(* IEC 61131-3 sources: SJ_AGV/PLC/Standard_functions.4.4.0/Autoload, 3 files *)

(* ---- AutoLoadFailCodes.TYP ---- *)
[IEC_IEC_NORM]
TYPE
	AutoLoadFailCodes_T:
		STRUCT
			FailCode_OK						: word	:= 16#0000;
			FailCode_AGV_HalfLoad			: word	:= 16#0001;		(* Load is on the forks, but not fully. Manual handling and reset required! *)
			FailCode_OPNoSupport 			: word	:= 16#0002;
			FailCode_OpCancel 				: word	:= 16#0004;
			FailCode_InvalidOP 				: word	:= 16#0008;
			FailCode_AGVIsLoaded 			: word	:= 16#0010;
			FailCode_STNIsEmpty 			: word	:= 16#0020;
			FailCode_AGVIsNotLoaded			: word	:= 16#0040;
			FailCode_STNIsFull 				: word	:= 16#0080;
			FailCode_FirstPalletTooHigh		: word	:= 16#0100;
			FailCode_NoSecondPallet			: word	:= 16#0200;
			FailCode_SecondPalletTooLow		: word	:= 16#0400;
			FailCode_PalletOnInitialLift	: word	:= 16#0800;
			FailCode_NoPalletOnInitialLift	: word	:= 16#1000;
			FailCode_BatteryCharge			: word	:= 16#2000;
		END_STRUCT;
END_TYPE

(* ---- AUTOLOAD_FB.ST ---- *)
FUNCTION_BLOCK AUTOLOAD_FB
VAR_EXTERNAL
	(* IN *)
	NDC8: NDC8_T;
END_VAR

VAR_INPUT
	ForkMoving	: bool;
	ForkTarget	: bool;
END_VAR

VAR

	(* BCD Process *)
	BCDProcState : dint;
	BCDRetryTimes : int := 5;
	BCDReCompTimes : int := 5;
	BCDReadTimes : int;
	BCDCompTimes : int;

	TempBCD1_Int : Int;
	TempBCD1 : Word;

	(* Load/Unload Process *)
	LoadOpDone : LoadOpDone_FB;
	OperationFail : OperationFail_FB;

	AutoLoadFailCodes : AutoLoadFailCodes_T;
	OperationCode	: word;

	AutoLoadMainState : dint;

	BbxTrig_FT : F_trig;
	ExecDriveCommand_RT : R_Trig;
	FailTimerTON : TON;

	PreviousMainState,
	PreviousLoadState,
	PreviousUnLoadState,
	PreviousTravelDir,
	PreviousFailCode,
	PreviousForkHeight,
	FailCodeDint : dint;

	PreviousExecDriveCommand,
	PreviousCancelOperation,
	bbxtrigger			:bool;

	StepDelay : TON;
	BCDStepDelay : TON;

	TempErrorCode : DINT;

	BCD_ReadReq : BOOL;

	DebugBCD_1000_F : BOOL := FALSE;
	DebugBCD_1000_B : BOOL := FALSE;

	Debug_1000_F : BOOL := FALSE;
	Debug_1000_B : BOOL:= FALSE;
	Debug_2000_F : BOOL:= FALSE;
	Debug_2000_B : BOOL:= FALSE;

	LrErrCode : DINT;

	(*Wait Barcode Answer 2s*)

	WiatBardCodeAnser : TON;
END_VAR

VAR_OUTPUT
	StartLoad : bool;
	StartUnload : bool;
	StartCharge	: bool;
	Fail : bool;
END_VAR
(*
------------------------------------------------------------------------------------
 AUTOLOAD_SD
 -----------

 Description:
 Handles load operations. Output is 'Fork height'.
 If there is a cancel, LoadOpDone will be sent to the host with a failcode.

-------------------------------------------------------------------------------------*)

(* Set up variables to be used from NDC8 sources *)
OperationCode 		:= dint_to_word(NDC8.LoadOperation.OperationCode);				(* Value is decimal in vehicle, but hex in Layout designer! *)

if (NDC8.Automatic.CurrentOrderMode = 2 or NDC8.Automatic.CurrentOrderMode = 3) and AutoloadMainState <> 2000 then (*in Local mode Operation code need to calcuate for PLC*)
		IN_OPCD_Bit_LT_Ang0		:= word_to_bool(OperationCode and 1);
		IN_OPCD_Bit_LT_Ang90	:= word_to_bool(OperationCode and 2);
		IN_OPCD_Bit_LT_Ang180	:= word_to_bool(OperationCode and 8);
		IN_OPCD_Bit_LT_AngN90	:= word_to_bool(OperationCode and 4);

		IN_OPCD_Bit_LT_Right	:= word_to_bool(OperationCode and 16);
		IN_OPCD_Bit_LT_Left		:= word_to_bool(OperationCode and 32);

		IN_OPCD_Bit_LT_Load 	:= word_to_bool(OperationCode and 256);
		IN_OPCD_Bit_LT_Unload	:= word_to_bool(OperationCode and 512);

		IN_OPCD_Bit_LT_PowOff	:= word_to_bool(OperationCode and 1024);
		IN_OPCD_Bit_LT_Charge	:= word_to_bool(OperationCode and 4096);

elsif NDC8.Automatic.CurrentOrderMode = 1 and AutoloadMainState <> 2000 then (*in Host mode Operation code need to calcuate for PLC*)
		IN_OPCD_Bit_LT_Ang0		:= word_to_bool(OperationCode and 16);
		IN_OPCD_Bit_LT_Ang90	:= word_to_bool(OperationCode and 32);
		IN_OPCD_Bit_LT_Ang180	:= word_to_bool(OperationCode and 64);
		IN_OPCD_Bit_LT_AngN90	:= word_to_bool(OperationCode and 128);

		IN_OPCD_Bit_LT_Right	:= word_to_bool(OperationCode and 1);
		IN_OPCD_Bit_LT_Left		:= word_to_bool(OperationCode and 2);

		IN_OPCD_Bit_LT_Load 	:= word_to_bool(OperationCode and 4096);
		IN_OPCD_Bit_LT_Unload	:= word_to_bool(OperationCode and 8192);

		IN_OPCD_Bit_Cmd_EnaEmg	:= word_to_bool(OperationCode and 256);

		IN_OPCD_Bit_LT_PowOff	:= word_to_bool(OperationCode and 16384);

		IN_OPCD_Bit_LT_Charge	:= word_to_bool(OperationCode and 32768);

else
		OperationCode := 0;
		InProc_OperationCode := 0;
end_if;

(*Check Str_EnaPB *)
if NDC8.OMPLC.Phase - 4 >= 0 then
	PLC_TX01_Bit_STr_EnaPB := TRUE;
else
	PLC_TX01_Bit_STr_EnaPB := FALSE;
end_if;

(* BCD Process *)
if NDC8.Automatic.CurrentOrderMode = 1 and PLC_RX01_Bit_Load_i = TRUE then

	case BCDProcState of
	0: (* Check BCD Req *)
		OM_PLC_Word2 := INT_TO_WORD(NDC8.OMPLC.Stop_OM);

		BCDReadTimes := 0;
		BCDCompTimes := 0;

		if BCD_ReadReq = TRUE and OM_PLC_W2_Bit_BCD_NoRead = FALSE then
			BCDProcState := 1;
		elsif BCD_ReadReq = TRUE and OM_PLC_W2_Bit_BCD_NoRead = TRUE then
			BCD_ReadReq := FALSE;
		elsif OM_PLC_W2_Bit_BCD_NoRead = TRUE then
			BCDProcState := 0;
		elsif OM_PLC_W2_Bit_BCD_Init = TRUE and OM_PLC_W2_Bit_BCD_NoRead = FALSE then
			BCDProcState := 1;
		elsif OM_PLC_W2_Bit_BCD_setReq = TRUE and OM_PLC_W2_Bit_BCD_NoRead = FALSE then
			BCDProcState := 1;
		end_if;

		NDC8.OMPLC.Stop_OM := WORD_TO_INT(OM_PLC_Word2);
	1: (*Clear BCD Req*)
		StopByBCD := TRUE;
		PLC_TX04_Bit_BCD_Clr := true;
		PLC_TX04_Bit_BCD_Req := false;

		OM_PLC_Word2 := INT_TO_WORD(NDC8.OMPLC.Stop_OM);
			OM_PLC_W2_Bit_BCD_setOK := FALSE;
			OM_PLC_W2_Bit_Set_Result := FALSE;
			OM_PLC_W2_Bit_Err_Comp := FALSE;
			OM_PLC_W2_Bit_Err_BCR := FALSE;
		NDC8.OMPLC.Stop_OM := WORD_TO_INT(OM_PLC_Word2);

		if	not PLC_RX06_Bit_BCD_OK
			and not PLC_RX06_Bit_NoRead_NG
			and not PLC_RX06_Bit_BCRHard_NG
			and not PLC_RX06_Bit_BCRData_NG
			and not PLC_RX06_Bit_BCRInit_NG
			and not PLC_RX06_Bit_BCRComm_NG then

			BCDProcState := 2;
		end_if;

	2: (*Set BCD Req*)
		PLC_TX04_Bit_BCD_Clr := false;
		PLC_TX04_Bit_BCD_Req := true;
		WiatBardCodeAnser(IN := PLC_TX04_Bit_BCD_Req , PT:= t#2s);
		BCDReadTimes := BCDReadTimes + 1;
	IF WiatBardCodeAnser.Q = TRUE THEN
		if PLC_RX06_Bit_BCD_OK
			and not PLC_RX06_Bit_NoRead_NG
			and not PLC_RX06_Bit_BCRHard_NG
			and not PLC_RX06_Bit_BCRData_NG
			and not PLC_RX06_Bit_BCRInit_NG
			and not PLC_RX06_Bit_BCRComm_NG then
			BCDReadTimes := 0;

			BCDProcState := 3;

		elsif 	PLC_RX06_Bit_NoRead_NG
				or PLC_RX06_Bit_BCRHard_NG
				or PLC_RX06_Bit_BCRData_NG
				or PLC_RX06_Bit_BCRInit_NG
				or PLC_RX06_Bit_BCRComm_NG then

			if BCDReadTimes >= BCDRetryTimes then
				OM_PLC_Word2 := INT_TO_WORD(NDC8.OMPLC.Stop_OM);
					OM_PLC_W2_Bit_Err_BCR := TRUE;
					OM_PLC_W2_Bit_Set_Result := TRUE;
				NDC8.OMPLC.Stop_OM := WORD_TO_INT(OM_PLC_Word2);
				BCDProcState := 1000;
			else
				BCDProcState := 1;
			end_if;
		end_if;
	END_IF;
	3: (*BCD Compare*)
		WiatBardCodeAnser(IN := FALSE);
		TempBCD1_Int := WORD_TO_INT(PLC_RX_Word9_STw_BCD1);(* - 16#D00*);
		TempBCD1 := INT_TO_WORD(TempBCD1_Int);

		BCDCompTimes := BCDCompTimes + 1;

		if 	PLC_TX_Word14_STr_BCD3 = PLC_RX_Word7_STw_BCD3
			and PLC_TX_Word15_STr_BCD2 = PLC_RX_Word8_STw_BCD2
			and PLC_TX_Word16_STr_BCD1 = PLC_RX_Word9_STw_BCD1 then
			BCDProcState := 4; (* Compare Complete *)
			BCDCompTimes := 0;

		else

			if BCDCompTimes >= BCDReCompTimes then
				OM_PLC_Word2 := INT_TO_WORD(NDC8.OMPLC.Stop_OM);
					OM_PLC_W2_Bit_Err_Comp := TRUE;
					OM_PLC_W2_Bit_Set_Result := TRUE;
				NDC8.OMPLC.Stop_OM := WORD_TO_INT(OM_PLC_Word2);
				BCDProcState := 1000;
			else
				BCDProcState := 1;
			end_if;

		end_if;

	4:
		OM_PLC_Word2 := INT_TO_WORD(NDC8.OMPLC.Stop_OM);
			OM_PLC_W2_Bit_BCD_setOK := TRUE;
			OM_PLC_W2_Bit_Set_Result := TRUE;
		NDC8.OMPLC.Stop_OM := WORD_TO_INT(OM_PLC_Word2);
		BCDProcState := 1000;

	1000: (*Reset*)

		if DebugBCD_1000_F = FALSE then
			if DebugBCD_1000_B = FALSE then
				BCDProcState := 0;
			end_if;
			BCDReadTimes := 0;
			BCDCompTimes := 0;

			BCD_ReadReq := FALSE;
			StopByBCD := FALSE;
			BCDStepDelay(IN:= FALSE);

			OM_PLC_Word2 := INT_TO_WORD(NDC8.OMPLC.Stop_OM);
				OM_PLC_W2_Bit_BCD_setReq := FALSE;
				OM_PLC_W2_Bit_BCD_Init := FALSE;
			NDC8.OMPLC.Stop_OM := WORD_TO_INT(OM_PLC_Word2);
		end_if;

	end_case;
end_if;

Case AutoloadMainState of

(**** Wait for AutoLoad Start Flag - Operation Code > 0 ****)
	0:

		OM_PLC_Word2 := INT_TO_WORD(NDC8.OMPLC.Stop_OM);

		PLC_TX_Word2 := 0;

		PLC_TX02_Bit_STr_DepoST := FALSE;
		PLC_TX02_Bit_STr_ShutEQ := FALSE;
		PLC_TX04_Bit_Cancel_ST := FALSE;
		StepDelay(IN := FALSE);
		if g_ErrorCode = 0 and PLC_RX01_Bit_EnableLD_i = TRUE then
			if OperationCode > 0 then
				AutoloadMainState := 10;
			elsif NDC8.LocalOrder.OrderEN then
				AutoloadMainState := 10;
			end_if;
		end_if;

(**** Load operations ****)
	10:
		BCD_ReadReq := FALSE;
		INPUT.AutoLoadDone := FALSE;
		if 	IN_OPCD_Bit_LT_Load then	(* Load *)
			AutoloadMainState := 20;
		elsif 	IN_OPCD_Bit_LT_Unload then	(* Unload *)
			AutoloadMainState := 30;
		elsif 	IN_OPCD_Bit_LT_Charge then	(* Charge battery *)
			AutoloadMainState := 40;
		elsif	IN_OPCD_Bit_LT_PowOff then	(* Power off *)
			AutoloadMainState := 50;
		elsif NDC8.LocalOrder.OpCode = 0 then
			AutoloadMainState := 60;		(* Move no OP Code *)
		end_if;

(* Pick up load *)
	20:	(*Check Vehicle on Target Station*)

		OM_PLC_Word2 := INT_TO_WORD(NDC8.OMPLC.Stop_OM);

			OM_PLC_W2_Bit_SetT10Terr := FALSE;
			OM_PLC_W2_Bit_SetCondErr := FALSE;
			OM_PLC_W2_Bit_SetT30TErr := FALSE;
			OM_PLC_W2_Bit_SetHOErr := FALSE;

		NDC8.OMPLC.Stop_OM := WORD_TO_INT(OM_PLC_Word2);

		if g_ErrorCode <> 0 then
			AutoloadMainState := 999;
		else
			StartLoad := true;
			if NDC8.LoadDocking.OnTarget = TRUE and PLC_RX01_Bit_EnableLD_i = TRUE then
				AutoloadMainState := 21;
			elsif NDC8.LoadDocking.OnTarget = TRUE and PLC_RX01_Bit_EnableLD_i = FALSE then
				AutoloadMainState := 148;
			elsif InProc_OperationCode = 0 then
				AutoloadMainState := 145;
			end_if;
		end_if;

	21:(*Check Robot Load status*)
		StopLoadOP := TRUE;
		if g_ErrorCode <> 0 then
			AutoloadMainState := 999;
		else
			if PLC_RX01_Bit_Load_i = true then
				AutoloadMainState := 148;
			elsif NDC8.SDIO.DigitalInput12_EMO = FALSE then
				AutoloadMainState := 133;
			else
				AutoloadMainState := 22;
			end_if;
		end_if;

	22:(*Set OpCode to PLC*)

		if g_ErrorCode <> 0 then
			AutoloadMainState := 999;
		else
			PLC_TX02_Bit_STr_Ang0	:= IN_OPCD_Bit_LT_Ang0;
			PLC_TX02_Bit_STr_Ang90	:= IN_OPCD_Bit_LT_Ang90;
			PLC_TX02_Bit_STr_Ang180	:= IN_OPCD_Bit_LT_Ang180;
			PLC_TX02_Bit_STr_AngN90	:= IN_OPCD_Bit_LT_AngN90;

			PLC_TX02_Bit_STr_Right	:= IN_OPCD_Bit_LT_Right;
			PLC_TX02_Bit_STr_Left	:= IN_OPCD_Bit_LT_Left;

			PLC_TX02_Bit_STr_Load 	:= IN_OPCD_Bit_LT_Load;
			PLC_TX02_Bit_STr_Unload	:= IN_OPCD_Bit_LT_Unload;

			PLC_TX02_Bit_STr_DepoST := NDC8.PointTrigger.Bit0_DepoST_Att;
			PLC_TX02_Bit_STr_ShutEQ := NDC8.PointTrigger.Bit1_ShutEQ_Att;
			PLC_TX04_Bit_Cancel_ST := not IN_OPCD_Bit_Cmd_EnaEmg;

			if (PLC_TX02_Bit_STr_Ang0 = TRUE and PLC_TX02_Bit_STr_Ang90 = TRUE)
				or (PLC_TX02_Bit_STr_Ang0 = TRUE and PLC_TX02_Bit_STr_Ang180 = TRUE)
				or (PLC_TX02_Bit_STr_Ang0 = TRUE and PLC_TX02_Bit_STr_AngN90 = TRUE)
				or (PLC_TX02_Bit_STr_Ang90 = TRUE and PLC_TX02_Bit_STr_Ang180 = TRUE)
				or (PLC_TX02_Bit_STr_Ang90 = TRUE and PLC_TX02_Bit_STr_AngN90 = TRUE)
				or (PLC_TX02_Bit_STr_Ang180 = TRUE and PLC_TX02_Bit_STr_AngN90 = TRUE)
				or (PLC_TX02_Bit_STr_Right = TRUE and PLC_TX02_Bit_STr_Left = TRUE)
				or (PLC_TX02_Bit_STr_Load = TRUE and PLC_TX02_Bit_STr_Unload = TRUE) then

				if NDC8.Automatic.CurrentOrderMode = 1 then
					AutoloadMainState := 150;
				elsif NDC8.Automatic.CurrentOrderMode = 2 or NDC8.Automatic.CurrentOrderMode = 3 then
					AutoloadMainState := 152;
				end_if;

			elsif 	PLC_TX02_Bit_STr_Ang0 = FALSE
					and PLC_TX02_Bit_STr_Ang90 = FALSE
					and PLC_TX02_Bit_STr_Ang180 = FALSE
					and PLC_TX02_Bit_STr_AngN90 = FALSE then
					AutoloadMainState := 145;

			elsif	PLC_TX02_Bit_STr_Right = FALSE
					and PLC_TX02_Bit_STr_Left = FALSE then
					AutoloadMainState := 145;

			elsif	PLC_TX02_Bit_STr_Load = FALSE
					and PLC_TX02_Bit_STr_Unload = FALSE then
					AutoloadMainState := 145;

			else
				AutoloadMainState := 23;
			end_if;
		end_if;

	23:(*Wait PLC Processing*)
		if g_ErrorCode <> 0 then
			AutoloadMainState := 999;
		else
			if INPUT.Auto = FALSE then
				AutoloadMainState := 998;
			elsif NDC8.SDIO.DigitalInput12_EMO = FALSE then
				AutoloadMainState := 133;
			elsif PLC_RX01_Bit_LDErr_i then
				AutoloadMainState := 148;
			elsif PLC_RX_Word10_STw_ILEr <> 0 then (* Interlock (8I/8O) Proc *)

				OM_PLC_Word2 := INT_TO_WORD(NDC8.OMPLC.Stop_OM);

				case PLC_RX_Word10_STw_ILEr of
				1:
					OM_PLC_W2_Bit_SetT10Terr := TRUE;
					AutoloadMainState := 900;
				2:
					OM_PLC_W2_Bit_SetCondErr := TRUE;
					AutoloadMainState := 900;
				3:
					OM_PLC_W2_Bit_SetT30TErr := TRUE;
					AutoloadMainState := 900;
				4:
					OM_PLC_W2_Bit_SetHOErr := TRUE;
					AutoloadMainState := 900;
				5:
					OM_PLC_W2_Bit_SetHOErr := TRUE;
					AutoloadMainState := 900;

				end_case;

				NDC8.OMPLC.Stop_OM := WORD_TO_INT(OM_PLC_Word2);

			elsif PLC_RX01_Bit_LDDone_i then
				PLC_TX_Word2 := 0;
				PLC_TX02_Bit_STr_DepoST := FALSE;
				PLC_TX02_Bit_STr_ShutEQ := FALSE;
				PLC_TX04_Bit_Cancel_ST := FALSE;
			IF NDC8.Automatic.CurrentOrderMode = 1 THEN
				StopByBCD := TRUE;
			END_IF;
				BCD_ReadReq := TRUE;

				AutoloadMainState := 1000;
			end_if;
		end_if;

(* Drop off load *)
	30:	(*Check Vehicle on Target Station*)

		OM_PLC_Word2 := INT_TO_WORD(NDC8.OMPLC.Stop_OM);

			OM_PLC_W2_Bit_SetT10Terr := FALSE;
			OM_PLC_W2_Bit_SetCondErr := FALSE;
			OM_PLC_W2_Bit_SetT30TErr := FALSE;
			OM_PLC_W2_Bit_SetHOErr := FALSE;

		NDC8.OMPLC.Stop_OM := WORD_TO_INT(OM_PLC_Word2);

		if g_ErrorCode <> 0 then
			AutoloadMainState := 999;
		else
			StartUnload := true;

			if NDC8.LoadDocking.OnTarget = TRUE and PLC_RX01_Bit_EnableLD_i = TRUE then
				AutoloadMainState := 31;
			elsif NDC8.LoadDocking.OnTarget = TRUE and PLC_RX01_Bit_EnableLD_i = FALSE then
				AutoloadMainState := 149;
			end_if;
		end_if;

	31:(*Check Robot Load status*)
		StopLoadOP := TRUE;

		if g_ErrorCode <> 0 then
			AutoloadMainState := 999;
		else
			if PLC_RX01_Bit_Load_i = false then
				AutoloadMainState := 149;
			elsif NDC8.SDIO.DigitalInput12_EMO = FALSE then
				AutoloadMainState := 133;
			else
				AutoloadMainState := 32;
			end_if;
		end_if;

	32: (*Set OpCode to PLC*)

		if g_ErrorCode <> 0 then
			AutoloadMainState := 999;
		else
			PLC_TX02_Bit_STr_Ang0	:= IN_OPCD_Bit_LT_Ang0;
			PLC_TX02_Bit_STr_Ang90	:= IN_OPCD_Bit_LT_Ang90;
			PLC_TX02_Bit_STr_Ang180	:= IN_OPCD_Bit_LT_Ang180;
			PLC_TX02_Bit_STr_AngN90	:= IN_OPCD_Bit_LT_AngN90;

			PLC_TX02_Bit_STr_Right	:= IN_OPCD_Bit_LT_Right;
			PLC_TX02_Bit_STr_Left	:= IN_OPCD_Bit_LT_Left;

			PLC_TX02_Bit_STr_Load 	:= IN_OPCD_Bit_LT_Load;
			PLC_TX02_Bit_STr_Unload	:= IN_OPCD_Bit_LT_Unload;

			PLC_TX02_Bit_STr_DepoST := NDC8.PointTrigger.Bit0_DepoST_Att;
			PLC_TX02_Bit_STr_ShutEQ := NDC8.PointTrigger.Bit1_ShutEQ_Att;

			PLC_TX04_Bit_Cancel_ST := not IN_OPCD_Bit_Cmd_EnaEmg;

			if (PLC_TX02_Bit_STr_Ang0 = TRUE and PLC_TX02_Bit_STr_Ang90 = TRUE)
				or (PLC_TX02_Bit_STr_Ang0 = TRUE and PLC_TX02_Bit_STr_Ang180 = TRUE)
				or (PLC_TX02_Bit_STr_Ang0 = TRUE and PLC_TX02_Bit_STr_AngN90 = TRUE)
				or (PLC_TX02_Bit_STr_Ang90 = TRUE and PLC_TX02_Bit_STr_Ang180 = TRUE)
				or (PLC_TX02_Bit_STr_Ang90 = TRUE and PLC_TX02_Bit_STr_AngN90 = TRUE)
				or (PLC_TX02_Bit_STr_Ang180 = TRUE and PLC_TX02_Bit_STr_AngN90 = TRUE)
				or (PLC_TX02_Bit_STr_Right = TRUE and PLC_TX02_Bit_STr_Left = TRUE)
				or (PLC_TX02_Bit_STr_Load = TRUE and PLC_TX02_Bit_STr_Unload = TRUE) then

				if NDC8.Automatic.CurrentOrderMode = 1 then
					AutoloadMainState := 150;
				elsif NDC8.Automatic.CurrentOrderMode = 2 or NDC8.Automatic.CurrentOrderMode = 3 then
					AutoloadMainState := 152;
				end_if;

			elsif 	PLC_TX02_Bit_STr_Ang0 = FALSE
					and PLC_TX02_Bit_STr_Ang90 = FALSE
					and PLC_TX02_Bit_STr_Ang180 = FALSE
					and PLC_TX02_Bit_STr_AngN90 = FALSE then
					AutoloadMainState := 145;

			elsif	PLC_TX02_Bit_STr_Right = FALSE
					and PLC_TX02_Bit_STr_Left = FALSE then
					AutoloadMainState := 145;

			elsif	PLC_TX02_Bit_STr_Load = FALSE
					and PLC_TX02_Bit_STr_Unload = FALSE then
					AutoloadMainState := 145;

			else
				AutoloadMainState := 33;
			end_if;
		end_if;

	33: (*Wait PLC Processing*)
		if g_ErrorCode <> 0 then
				AutoloadMainState := 999;
		else
			if INPUT.Auto = FALSE then
				AutoloadMainState := 998;
			elsif NDC8.SDIO.DigitalInput12_EMO = FALSE then
				AutoloadMainState := 133;
			elsif PLC_RX01_Bit_LDErr_i then
				AutoloadMainState := 149;
			elsif PLC_RX_Word10_STw_ILEr <> 0 then (* Interlock (8I/8O) Proc *)

				OM_PLC_Word2 := INT_TO_WORD(NDC8.OMPLC.Stop_OM);

				case PLC_RX_Word10_STw_ILEr of
				1:
					OM_PLC_W2_Bit_SetT10Terr := TRUE;
					AutoloadMainState := 900;
				2:
					OM_PLC_W2_Bit_SetCondErr := TRUE;
					AutoloadMainState := 900;
				3:
					OM_PLC_W2_Bit_SetT30TErr := TRUE;
					AutoloadMainState := 900;
				4:
					OM_PLC_W2_Bit_SetHOErr := TRUE;
					AutoloadMainState := 900;
				5:
					OM_PLC_W2_Bit_SetHOErr := TRUE;
					AutoloadMainState := 900;

				end_case;

				NDC8.OMPLC.Stop_OM := WORD_TO_INT(OM_PLC_Word2);

			elsif PLC_RX01_Bit_LDDone_i then
				PLC_TX_Word2 := 0;
				PLC_TX02_Bit_STr_DepoST := FALSE;
				PLC_TX02_Bit_STr_ShutEQ := FALSE;
				PLC_TX04_Bit_Cancel_ST := FALSE;
				AutoloadMainState := 1000;
			end_if;
		end_if;

(* Charge the battery Local Order *)
	40:
		if g_ErrorCode <> 0 then
			AutoloadMainState := 999;
		else
			if NDC8.LoadDocking.OnTarget = TRUE then
				(* Wait Charger InPosition *)

				(* Check Charge Idle*)
				if PLC_RX01_Bit_ChrgIdle then
					AutoloadMainState := 41;
				end_if;

			end_if;
		end_if;

	41:(* Check OpCode and wait 10sec*)

		if g_ErrorCode <> 0 then
			AutoloadMainState := 49;
		else
			if INPUT.Auto = FALSE then
				AutoloadMainState := 49;
			end_if;

			if NDC8.PointTrigger.Bit9_Chrg_Right = TRUE or NDC8.PointTrigger.Bit10_Chrg_Left = TRUE  then
				StopCharge := TRUE;

				OM_PLC_Word2 := INT_TO_WORD(NDC8.OMPLC.Stop_OM);

				if (NDC8.Automatic.CurrentOrderMode = 1 and OM_PLC_W2_Bit_Set_LowTS) or NDC8.Automatic.CurrentOrderMode <> 1 then
					AutoloadMainState := 42;
				end_if;
			else
				;(*OP Error*)
			end_if;
		end_if;

	42:

		if g_ErrorCode <> 0 then
			AutoloadMainState := 49;
		else
			if INPUT.Auto = FALSE then
				AutoloadMainState := 49;
			end_if;
			IF NDC8.PointTrigger.Bit9_Chrg_Right = TRUE and NDC8.PointTrigger.Bit10_Chrg_Left = FALSE  then
				PLC_TX04_Bit_ChrgCmdR_A := TRUE;
				PLC_TX04_Bit_ChrgCmdL_A := FALSE;
				NDC8.SDIO.DigitalOutput16_RIGHTMGS := TRUE;
			END_IF;

			IF NDC8.PointTrigger.Bit9_Chrg_Right = FALSE and NDC8.PointTrigger.Bit10_Chrg_Left = TRUE  then
				PLC_TX04_Bit_ChrgCmdL_A := TRUE;
				PLC_TX04_Bit_ChrgCmdR_A := FALSE;
				NDC8.SDIO.DigitalOutput12_LEFTMGS := TRUE;
			END_IF;

			OM_PLC_Word2 := INT_TO_WORD(NDC8.OMPLC.Stop_OM);

			if (NDC8.Automatic.CurrentOrderMode = 1 and OM_PLC_W2_Bit_Set_LowTS = false) or (g_ErrorCode <> 0 or PLC_RX15_Bit_BMS_ChgCmp or PLC_RX01_Bit_ChrgEmg) then
				AutoloadMainState := 43;
			end_if;
		end_if;

	43:

		if g_ErrorCode <> 0 then
			AutoloadMainState := 49;
		else
			if INPUT.Auto = FALSE then
				AutoloadMainState := 49;
			end_if;

			PLC_TX04_Bit_ChrgCmdL_A := FALSE;

			PLC_TX04_Bit_ChrgCmdR_A := FALSE;

			NDC8.SDIO.DigitalOutput16_RIGHTMGS := FALSE;

			NDC8.SDIO.DigitalOutput12_LEFTMGS := FALSE;

			OM_PLC_Word1 := INT_TO_WORD(NDC8.OMPLC.ChargeOM);

			OM_PLC_W1_Bit_SetLowBatt := FALSE;

			NDC8.OMPLC.ChargeOM := WORD_TO_INT(OM_PLC_Word1);

			if PLC_RX01_Bit_ChrgIdle then
				StepDelay(IN:=TRUE, PT:=t#1s);
				if StepDelay.Q then
					StepDelay(IN:=FALSE);
					AutoloadMainState := 1000;
					StopCharge := FALSE;
				end_if;
			end_if;

		end_if;

	49:

		PLC_TX04_Bit_ChrgCmdL_A := FALSE;

		PLC_TX04_Bit_ChrgCmdR_A := FALSE;

		NDC8.SDIO.DigitalOutput16_RIGHTMGS := FALSE;

		NDC8.SDIO.DigitalOutput12_LEFTMGS := FALSE;

		OM_PLC_Word1 := INT_TO_WORD(NDC8.OMPLC.ChargeOM);

		OM_PLC_W1_Bit_SetLowBatt := FALSE;

		NDC8.OMPLC.ChargeOM := WORD_TO_INT(OM_PLC_Word1);

		if PLC_RX01_Bit_ChrgIdle then
			StepDelay(IN:=TRUE, PT:=t#1s);
			if StepDelay.Q then
				StepDelay(IN:=FALSE);
				StopCharge := FALSE;

				if g_ErrorCode <> 0 then
					AutoloadMainState := 999;
				end_if;

				if INPUT.Auto = FALSE then
					AutoloadMainState := 998;
				end_if;

			end_if;
		end_if;

(* Power Off *)
	50:
		if g_ErrorCode <> 0 then
			AutoloadMainState := 999;
		else
			(* Send Event *)
			if NDC8.LoadDocking.OnTarget = TRUE then
				g_PowerOffFlag_OP := TRUE;
				if NDC8.SDIO.DigitalOutput13_PWR_OFF = TRUE then
					AutoloadMainState := 1000;
				end_if;
			end_if;
		end_if;

(* Move no OP Code *)
	60:
		if g_ErrorCode <> 0 then
			AutoloadMainState := 999;
		else
			StepDelay(IN := TRUE, PT := t#5s);

			if StepDelay.Q then
				if NDC8.LayoutPosition.Point = NDC8.LocalOrder.DestPoint then
					AutoloadMainState := 1000;
					StepDelay(IN := FALSE);
				end_if;

			end_if;
		end_if;

(* EMO *)
	133:
		g_ErrorCode := 133;
		Fail := TRUE;

		StepDelay(IN := TRUE, PT := t#1s);

		if StepDelay.Q then
			if NDC8.SDIO.DigitalInput12_EMO = TRUE then
				AutoloadMainState := 2000;
			end_if;
			StepDelay(IN := FALSE);
		end_if;

(* Transfer Schedule Error *)
	145:
		g_ErrorCode := 145;
		Fail := TRUE;

		StepDelay(IN := TRUE, PT := t#1s);

		if StepDelay.Q then
			AutoloadMainState := 2000;
			StepDelay(IN := FALSE);
		end_if;

(* Load Condition Error *)
	147:

		Fail := TRUE;

		StepDelay(IN := TRUE, PT := t#1s);

		if StepDelay.Q then
			AutoloadMainState := 2000;
			StepDelay(IN := FALSE);
		end_if;

(* Loading Condition Error *)
	148:
		g_ErrorCode := 148;
		Fail := TRUE;

		StepDelay(IN := TRUE, PT := t#1s);

		if StepDelay.Q then
			AutoloadMainState := 2000;
			StepDelay(IN := FALSE);
		end_if;

(* Unloading Condition Error *)
	149:

		Fail := TRUE;
		g_ErrorCode := 149;
		StepDelay(IN := TRUE, PT := t#1s);

		if StepDelay.Q then
			AutoloadMainState := 2000;
			StepDelay(IN := FALSE);
		end_if;

(* Command Error *)
	150:
		g_ErrorCode := 150;
		Fail := TRUE;

		StepDelay(IN := TRUE, PT := t#1s);

		if StepDelay.Q then
			AutoloadMainState := 2000;
			StepDelay(IN := FALSE);
		end_if;

(* Local Command Error *)
	152:
		g_ErrorCode := 152;
		Fail := TRUE;

		StepDelay(IN := TRUE, PT := t#1s);

		if StepDelay.Q then
			AutoloadMainState := 2000;
			StepDelay(IN := FALSE);
		end_if;

(* Ir Error Need to Error Stop Order  *)
	900:
		Fail := TRUE;

		if OM_PLC_W2_Bit_SetT10Terr = TRUE then
			LrErrCode := 243;
		elsif OM_PLC_W2_Bit_SetCondErr = TRUE then
			LrErrCode := 242;
		elsif OM_PLC_W2_Bit_SetT30TErr = TRUE then
			LrErrCode := 245;
		elsif OM_PLC_W2_Bit_SetHOErr = TRUE then
			LrErrCode := 259;
		elsif OM_PLC_W2_Bit_SetHOErr = TRUE then
			LrErrCode := 260;
		end_if;

		StepDelay(IN := TRUE, PT := t#1s);

		if StepDelay.Q then
			LoadOpDone(ErrorCode:=LrErrCode, Result:=NDC8.LayoutPosition.Distance);	(* Operation Fail Error=149 *)
			if LoadOpDone.Finished then
				INPUT.AutoLoadDone := TRUE;
				StopLoadOP := FALSE;
				AutoloadMainState:= 2000;	(* End autoload *)
			end_if;
		end_if;

(* Change Mode to Manual don't stop Order *)
	998:
		Fail := TRUE;

		StepDelay(IN := TRUE, PT := t#1s);

		if StepDelay.Q then
			AutoloadMainState := 2000;
			StepDelay(IN := FALSE);
		end_if;

(* Other Error Code Ocuur  don't stop Order *)
	999:

		Fail := TRUE;

		StepDelay(IN := TRUE, PT := t#1s);

		if StepDelay.Q then
			AutoloadMainState := 2000;
			StepDelay(IN := FALSE);
		end_if;

(**** Check if Operation Done OK ****)
	1000:

		if Debug_1000_F = FALSE then
			LoadOpDone(ErrorCode:=0, Result:=NDC8.LayoutPosition.Distance);	(* Operation OK Error=0 *)
			if LoadOpDone.Finished then
				Fail := FALSE;
				INPUT.AutoLoadDone := TRUE;
				StopLoadOP := FALSE;

				if Debug_1000_B = FALSE then
					AutoloadMainState:= 2000;	(* End autoload *)
				end_if;
			end_if;
		end_if;

(* Operation Complete *)
	2000:
		(*NDC8.LoadOperation.OperationCode := 0;
		InProc_OperationCode			:= 0;*)
		if Debug_2000_F = FALSE then
			if INPUT.AutoLoadDone = TRUE THEN
				StartLoad 						:= false;
				StartUnLoad 					:= false;
				StartCharge						:= false;

				InProc_OperationCode			:= 0;
				PLC_TX_Word2 := 0;

				StepDelay(IN := TRUE, PT := t#1s);

				if StepDelay.Q then
					AutoloadMainState := 2000;

					if Debug_2000_B = FALSE then
						AutoloadMainState				:= 0;
					end_if;

					StepDelay(IN := FALSE);
				end_if;

			else
				if Input.Manual = TRUE or g_AGV_ErrorReset = TRUE then
					INPUT.AutoLoadDone := TRUE;
					StopLoadOP := FALSE;
					AutoloadMainState				:= 0;
				end_if;
			end_if;
		end_if;
end_case;

(*===============================================*)
(* 		DEBUG #0x1  	Event 801				 *)

if word_to_bool(int_to_word(ndc8.omplc.DebugLevel) and 16#01) then
	if  debug or
		(PreviousMainState 						<> AutoLoadMainState) or
		(PreviousExecDriveCommand 				<> NDC8.Automatic.ExecDriveCommand) or
		(PreviousFailCode 						<> FailCodeDint) or
		(PreviousCancelOperation 				<> NDC8.LoadOperation.CancelOperation) or
		(PreviousTravelDir					 	<> NDC8.VehicleControl.TravelDir)
			then
				a:= TRACE_DINT('ALState',AutoLoadMainState);
				a:= TRACE_DINT('FailCodeDint',FailCodeDint);

				debug := true;
	end_if;
	PreviousExecDriveCommand 				:= NDC8.Automatic.ExecDriveCommand;
	PreviousTravelDir					 	:= NDC8.VehicleControl.TravelDir;
	PreviousMainState 						:= AutoloadMainState;
	PreviousFailCode						:= FailCodeDint;
	PreviousCancelOperation					:= NDC8.LoadOperation.CancelOperation;
	bbxtrigger:= AutoloadMainState=99 ;
	BbxTrig_FT(CLK:=bbxtrigger);
end_if;

(* If trigger do a blackbox and log event*)
if BbxTrig_FT.q then
	a:=TRACE_string('Bbx_Autoload');
	a:=TRACE_bool('BbxTrig',BbxTrig);
	NDC8.BlackBox.TrigReason:= 'Autoload';
	BbxTrig:=true;
end_if;

(* OUTPUT *)

END_FUNCTION_BLOCK

(* ---- OPERATIONFAIL_FB.ST ---- *)
FUNCTION_BLOCK OPERATIONFAIL_FB
VAR_EXTERNAL
	(* IN *)
	NDC8: NDC8_T;

END_VAR

VAR
	Failstate:dINT;
	LoadOpDone:LoadOpDone_FB;
END_VAR

VAR_INPUT
	FailCode:DINT;
END_VAR

VAR_OUTPUT
	Finished:bool:=false;
END_VAR
(*
------------------------------------------------------------------------------------
 OPERATION FAIL
 -----------

 Description:
 	If load operation fails, fail code is sent to the stationary system.

-------------------------------------------------------------------------------------*)

case Failstate of
	0:	Failstate := 1;
		Finished:= false;

	1: 	(* Cancel and LoadOp Clean-up required *)
		if 	NDC8.LoadDocking.OnTarget
				or NDC8.VehicleControl.OperationMode <> 0
			then
				Failstate := 2;

		elsif NDC8.LoadOperation.OperationCode = 0 	then				(* will not reach OnTarget *)
																(* Cancel and LoadOp clean-up NOT required *)
				Failstate := 3;
		end_if;

	2:	(* Clean up LoadOp for cancel *)
		LoadOpDone(ErrorCode:=FailCode, Result:=NDC8.LayoutPosition.Distance);	(* Send failcode *)
		if LoadOpDone.Finished then 										(* Move on when LoadOp Done	*)
			Failstate := 3;
		end_if;

	3:	(* Cancel Comlpete, run handshake and reset cancel state *)
		Finished:= true;
		Failstate := 0;
end_case;

END_FUNCTION_BLOCK
